FUNCTION_BLOCK POU
VAR_INPUT
END_VAR
VAR_OUTPUT
END_VAR
VAR
END_VAR


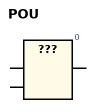
// PAGE
???(???, ???);

END_FUNCTION_BLOCK

(* stored: Version 1.1.0.1, ProductVersion 3.1.4018.5
   POU POU: Id {726e36f1-9c63-46c5-95db-fc50a15178b9}, SpecialFunc None *)
